// TwinCAT 3 PLC project Nepionic_OTel_IntegrationTest
// ProgramVersion: 3.1.4026.25
// libraries:
//   [Nepionic_Log], * (Nepionic)
//   Tc2_Standard, * (Beckhoff Automation GmbH)
//   Tc2_System, * (Beckhoff Automation GmbH)
//   Tc2_Utilities, * (Beckhoff Automation GmbH)
// project tree:
//   Lib/ Valve.TcPOU, FilterConfig.TcDUT, FilterSimulation.TcPOU, FilterState.TcDUT (not stored), Valve.TcPOU
//   Programs/ Main.TcPOU
//   Tasks/ PlcTask.TcTTO
// real-time tasks:
//   TASK PlcTask: cycle T#10ms, priority 20, ADS port 350

CONFIGURATION Nepionic_OTel_IntegrationTest
    RESOURCE PLC ON TwinCAT3
        TASK PlcTask(INTERVAL := T#10ms, PRIORITY := 20);
        PROGRAM Main WITH PlcTask : Main;
    END_RESOURCE
END_CONFIGURATION

// ---- Lib/FilterConfig.TcDUT
/// Configuration parameters for the sand filter simulation.
/// All *_s fields are in simulated seconds.
/// Real elapsed time = simulated_time / time_scale.
TYPE FilterConfig :
STRUCT
    /// Nominal (clean-filter) differential pressure across the filter bank (bar).
    dp_nominal_bar         : LREAL := 0.15;
    /// Differential pressure that triggers a backwash cycle (bar).
    dp_trigger_bar         : LREAL := 0.80;
    /// Theoretical maximum differential pressure of a fully blocked filter (bar).
    dp_max_bar             : LREAL := 1.40;
    /// Nominal pump flow rate during normal two-module filtering (L/min).
    flow_nominal_lpm       : LREAL := 500.0;
    /// Reduced pump flow rate during backwash — one module out of service (L/min).
    flow_backwash_lpm      : LREAL := 340.0;
    /// Static inlet pressure at nominal flow with a clean filter (bar).
    pressure_inlet_bar     : LREAL := 2.50;
    /// Simulated time for the filter to block from clean to dp_trigger_bar (seconds).
    blockage_time_s        : LREAL := 300.0;
    /// Duration of each individual module backwash phase (simulated seconds).
    backwash_duration_s    : LREAL := 30.0;
    /// Settling delay between Module A backwash end and Module B backwash start
    /// (simulated seconds).
    inter_backwash_delay_s : LREAL := 5.0;
    /// Post-backwash settling period before resuming normal filtering
    /// (simulated seconds).
    post_backwash_settle_s : LREAL := 10.0;
    /// Simulation time scale: simulated seconds that pass per real second.
    /// 10.0 means the filter blocks in blockage_time_s/10 real seconds.
    time_scale             : LREAL := 10.0;
    /// PLC task cycle time (ms) — used for per-scan blockage accumulation.
    cycle_time_ms          : LREAL := 10.0;
END_STRUCT
END_TYPE

// ---- Programs/Main.TcPOU
/// Integration test: self-cleaning reverse-flow sand filter.
///
/// Wires the FilterSimulation to the Nepionic Log + Metrics OTel bridge.
/// Both the log ring and metric ring are exposed as ADS symbols — point
/// the otelcol-ads collector at:
///   Logs    : Main.log_appender.ring
///   Metrics : Main.metric_ring
PROGRAM Main
VAR
    // ── OTel log backend ───────────────────────────────────────────────────────
    log_appender : Nepionic_Log_OTel.OTelLogAppender;

    // ── OTel metrics backend ───────────────────────────────────────────────────
    metric_core : Nepionic_Metrics_OTel.OTelMetricCore;

    // ── Application logger ─────────────────────────────────────────────────────
    logger : Nepionic_Log.DefaultLogger('SandFilter.Controller');

    // ── Filter simulation ──────────────────────────────────────────────────────
    config : FilterConfig;    // Uses DUT default values; tune at runtime.
    sim : FilterSimulation;

    // ── Metric publish interval (real time, independent of sim time_scale) ─────
    metric_timer : TON;

    // ── One-shot initialisation guard ─────────────────────────────────────────
    initialised : BOOL;

    // ── Metric attribute scratch buffers ──────────────────────────────────────
    m_attrs : ARRAY[0..4] OF Nepionic_Metrics.MetricAttribute;
    m_empty : ARRAY[0..4] OF Nepionic_Metrics.MetricAttribute;
	
	trigger_div_zero : BOOL;
	_div_zero : FLOAT;
	
	heartbeat_timer : TOn;
END_VAR

// ── One-time initialisation ───────────────────────────────────────────────────
IF NOT initialised THEN
    Nepionic_Log.GetLogManager().Register(log_appender);
    initialised := TRUE;
    logger.Info('Sand filter OTel integration test initialised');
END_IF

// ── Run filter simulation ─────────────────────────────────────────────────────
sim(Config := config);

// ── Log on state-transition events ───────────────────────────────────────────
// DP threshold crossed — backwash is about to begin.
IF sim.EvFilterBlocked THEN
    logger
        .WithAttribute('state', 'Filtering')
        .Warning('Differential pressure exceeded backwash threshold - scheduling backwash cycle');
END_IF

// Module A backwash valve just opened.
IF sim.EvBackwashStartedA THEN
    logger
        .WithAttribute('module', 'A')
        .WithAttribute('valve',  'reverse_flow_A')
        .Info('Backwash started - Module A reverse-flow valve open, waste port active');
END_IF

// Module B backwash valve just opened.
IF sim.EvBackwashStartedB THEN
    logger
        .WithAttribute('module', 'B')
        .WithAttribute('valve',  'reverse_flow_B')
        .Info('Backwash started - Module B reverse-flow valve open, waste port active');
END_IF

// Both modules cleaned; filter bank back in service.
IF sim.EvBackwashComplete THEN
    logger
        .WithAttribute('cycles_completed', UDINT_TO_STRING(sim.BackwashCycles))
        .Info('Full backwash cycle complete - both modules clean, differential pressure at nominal');
END_IF

// ── Publish metrics every second (real time) ──────────────────────────────────
metric_timer(IN := TRUE, PT := T#1S);
IF metric_timer.Q THEN
    metric_timer(IN := FALSE); // reset for next interval

    // Pump flow
    metric_core.Record(
        'filter.flow_rate', 'L/min',
        sim.PumpFlowLpm,
        Nepionic_Metrics.MetricKind.Gauge, m_empty, 0);

    // Filter bank pressures
    metric_core.Record(
        'filter.pressure.inlet', 'bar',
        sim.PressureInletBar,
        Nepionic_Metrics.MetricKind.Gauge, m_empty, 0);

    metric_core.Record(
        'filter.pressure.outlet', 'bar',
        sim.PressureOutletBar,
        Nepionic_Metrics.MetricKind.Gauge, m_empty, 0);

    metric_core.Record(
        'filter.pressure.differential', 'bar',
        sim.DpBar,
        Nepionic_Metrics.MetricKind.Gauge, m_empty, 0);

    // Blockage fraction — key indicator driving the backwash trigger
    metric_core.Record(
        'filter.blockage_fraction', '1',
        sim.BlockageFraction,
        Nepionic_Metrics.MetricKind.Gauge, m_empty, 0);

    // Monotonically increasing backwash cycle counter
    metric_core.Record(
        'filter.backwash.cycles_total', '{cycles}',
        UDINT_TO_LREAL(sim.BackwashCycles),
        Nepionic_Metrics.MetricKind.Counter, m_empty, 0);

    // Per-module backwash valve state (0=closed, 1=open), labelled by module
    m_attrs[0].key := 'module'; m_attrs[0].value := 'A';
    metric_core.Record(
        'filter.valve.backwash_active', '1',
        SEL(sim.ValveAOpen, 0.0, 1.0),
        Nepionic_Metrics.MetricKind.Gauge, m_attrs, 1);

    m_attrs[0].value := 'B';
    metric_core.Record(
        'filter.valve.backwash_active', '1',
        SEL(sim.ValveBOpen, 0.0, 1.0),
        Nepionic_Metrics.MetricKind.Gauge, m_attrs, 1);
END_IF

IF trigger_div_zero THEN
	trigger_div_zero := FALSE;
	_div_zero := 1 / _div_zero;
END_IF

heartbeat_timer(In := NOT heartbeat_timer.Q, PT := T#5S);
IF heartbeat_timer.Q THEN
    log_appender.Heartbeat();
	metric_core.Heartbeat();
END_IF

END_PROGRAM

// ---- Lib/FilterSimulation.TcPOU
/// Simulated reverse-flow self-cleaning sand filter with two filter modules.
///
/// Physical model
/// ─────────────
/// Filtering (normal):
///   Pump → Inlet → [Module A + Module B in parallel] → Outlet
///   Differential pressure rises as both modules accumulate blockage.
///
/// Backwash (Module A):
///   Clean outlet water is diverted backwards through Module A → Waste.
///   Module B carries all forward flow; DP reflects one module.
///
/// Backwash (Module B):  symmetric to Module A.
///
/// After BackwashB completes the blockage fraction is reset to zero and the
/// differential pressure returns to nominal.
///
/// Call every PLC scan and read the VAR_OUTPUT fields.
FUNCTION_BLOCK FilterSimulation
VAR_INPUT
    /// Simulation configuration (may be updated at runtime).
    Config : FilterConfig;
END_VAR
VAR_OUTPUT
    // ── Sensors ───────────────────────────────────────────────────────────────
    /// Pump flow rate (L/min).
    PumpFlowLpm         : LREAL;
    /// Filter bank inlet pressure (bar).
    PressureInletBar    : LREAL;
    /// Filter bank outlet pressure (bar).
    PressureOutletBar   : LREAL;
    /// Differential pressure across the filter bank: inlet − outlet (bar).
    DpBar               : LREAL;

    // ── Valve states ──────────────────────────────────────────────────────────
    /// TRUE when Module A reverse-flow backwash valve is open.
    ValveAOpen          : BOOL;
    /// TRUE when Module B reverse-flow backwash valve is open.
    ValveBOpen          : BOOL;

    // ── Status ────────────────────────────────────────────────────────────────
    /// Current controller state.
    State               : FilterState := FilterState.Filtering;
    /// Number of complete two-module backwash cycles executed since PLC start.
    BackwashCycles      : UDINT;
    /// Blockage fraction: 0.0 = completely clean, 1.0 = theoretical dp_max_bar.
    BlockageFraction    : LREAL;

    // ── Event pulses (TRUE for exactly one scan on the triggering transition) ─
    /// DP has just exceeded dp_trigger_bar — backwash is about to start.
    EvFilterBlocked     : BOOL;
    /// Module A backwash valve has just been opened.
    EvBackwashStartedA  : BOOL;
    /// Module B backwash valve has just been opened.
    EvBackwashStartedB  : BOOL;
    /// Full two-module backwash cycle just completed; blockage reset to zero.
    EvBackwashComplete  : BOOL;
END_VAR
VAR
    _blockage         : LREAL := 0.0;  // 0.0 (clean) → 1.0 (at dp_max_bar)
    _entry            : BOOL  := TRUE; // TRUE on the first scan of a new state
    _timer            : TON;
    _timer_pt         : TIME;
    _valveA           : Valve;
    _valveB           : Valve;
    _noise_t          : LREAL := 0.0;  // noise oscillator phase accumulator
    _noise            : LREAL;         // composite dimensionless noise signal
    _sim_dt           : LREAL;         // simulated seconds elapsed this scan
    _blockage_trigger : LREAL;         // blockage fraction that fires backwash
END_VAR

// ── Per-scan simulated timestep ──────────────────────────────────────────────
_sim_dt := Config.cycle_time_ms * 0.001 * Config.time_scale;

// Normalised blockage fraction at which dp_trigger_bar is reached.
_blockage_trigger := (Config.dp_trigger_bar - Config.dp_nominal_bar)
                   / (Config.dp_max_bar     - Config.dp_nominal_bar);

// ── Multi-frequency noise oscillator ─────────────────────────────────────────
// Phase advances at ~0.5 rad/real-second, giving a ~12-second noise period.
_noise_t := _noise_t + Config.cycle_time_ms * 0.001 * 0.5;
IF _noise_t > 628.0 THEN _noise_t := _noise_t - 628.0; END_IF
_noise := 0.015 * SIN(_noise_t)
        + 0.008 * SIN(_noise_t * 2.37 + 1.1)
        + 0.004 * SIN(_noise_t * 5.13 + 2.3);

// ── Clear event pulses ────────────────────────────────────────────────────────
EvFilterBlocked    := FALSE;
EvBackwashStartedA := FALSE;
EvBackwashStartedB := FALSE;
EvBackwashComplete := FALSE;

// ── State machine ─────────────────────────────────────────────────────────────
CASE State OF

    FilterState.Filtering:
        _valveA(Open := FALSE, Close := TRUE);
        _valveB(Open := FALSE, Close := TRUE);

        // Blockage accumulates while both modules are filtering.
        _blockage := MIN(_blockage + _sim_dt / Config.blockage_time_s, 1.0);

        // Trigger backwash when DP crosses dp_trigger_bar.
        IF _blockage >= _blockage_trigger THEN
            EvFilterBlocked := TRUE;
            State           := FilterState.BackwashA;
            _entry          := TRUE;
        END_IF

    FilterState.BackwashA:
        // Module A valve open: clean water from Module B flushes Module A to waste.
        _valveA(Open := TRUE,  Close := FALSE);
        _valveB(Open := FALSE, Close := TRUE);

        IF _entry THEN
            _entry             := FALSE;
            EvBackwashStartedA := TRUE;
            _timer(IN := FALSE, PT := T#0S); // reset
        ELSE
            _timer_pt := UDINT_TO_TIME(LREAL_TO_UDINT(
                Config.backwash_duration_s / Config.time_scale * 1000.0));
            _timer(IN := TRUE, PT := _timer_pt);
            IF _timer.Q THEN
                _timer(IN := FALSE, PT := T#0S);
                State  := FilterState.PauseBetween;
                _entry := TRUE;
            END_IF
        END_IF

    FilterState.PauseBetween:
        // Both valves closed; brief settling before opening Module B valve.
        _valveA(Open := FALSE, Close := TRUE);
        _valveB(Open := FALSE, Close := TRUE);

        IF _entry THEN
            _entry := FALSE;
            _timer(IN := FALSE, PT := T#0S);
        ELSE
            _timer_pt := UDINT_TO_TIME(LREAL_TO_UDINT(
                Config.inter_backwash_delay_s / Config.time_scale * 1000.0));
            _timer(IN := TRUE, PT := _timer_pt);
            IF _timer.Q THEN
                _timer(IN := FALSE, PT := T#0S);
                State  := FilterState.BackwashB;
                _entry := TRUE;
            END_IF
        END_IF

    FilterState.BackwashB:
        // Module B valve open: clean water from Module A flushes Module B to waste.
        _valveA(Open := FALSE, Close := TRUE);
        _valveB(Open := TRUE,  Close := FALSE);

        IF _entry THEN
            _entry             := FALSE;
            EvBackwashStartedB := TRUE;
            _timer(IN := FALSE, PT := T#0S);
        ELSE
            _timer_pt := UDINT_TO_TIME(LREAL_TO_UDINT(
                Config.backwash_duration_s / Config.time_scale * 1000.0));
            _timer(IN := TRUE, PT := _timer_pt);
            IF _timer.Q THEN
                _timer(IN := FALSE, PT := T#0S);
                _blockage := 0.0;  // Both modules cleaned — reset blockage.
                State     := FilterState.PostBackwash;
                _entry    := TRUE;
            END_IF
        END_IF

    FilterState.PostBackwash:
        // Both valves closed; pressure and flow settle before resuming filtering.
        _valveA(Open := FALSE, Close := TRUE);
        _valveB(Open := FALSE, Close := TRUE);

        IF _entry THEN
            _entry             := FALSE;
            EvBackwashComplete := TRUE;
            BackwashCycles     := BackwashCycles + 1;
            _timer(IN := FALSE, PT := T#0S);
        ELSE
            _timer_pt := UDINT_TO_TIME(LREAL_TO_UDINT(
                Config.post_backwash_settle_s / Config.time_scale * 1000.0));
            _timer(IN := TRUE, PT := _timer_pt);
            IF _timer.Q THEN
                _timer(IN := FALSE, PT := T#0S);
                State  := FilterState.Filtering;
                _entry := TRUE;
            END_IF
        END_IF

END_CASE

// ── Valve outputs ─────────────────────────────────────────────────────────────
ValveAOpen       := _valveA.IsOpen;
ValveBOpen       := _valveB.IsOpen;
BlockageFraction := _blockage;

// ── Differential pressure ─────────────────────────────────────────────────────
// During backwash one module is bypassed; DP reflects the remaining clean module
// (slightly above nominal due to full flow through half the filter area).
// During filtering the DP rises linearly with blockage, noised for realism.
IF    State = FilterState.BackwashA
   OR State = FilterState.PauseBetween
   OR State = FilterState.BackwashB THEN
    DpBar := Config.dp_nominal_bar * 1.25 * (1.0 + _noise);
ELSE
    DpBar := Config.dp_nominal_bar
           + _blockage * (Config.dp_max_bar - Config.dp_nominal_bar);
    DpBar := DpBar * (1.0 + _noise);
END_IF
DpBar := MAX(DpBar, 0.0);

// ── Inlet pressure ────────────────────────────────────────────────────────────
// The pump works slightly harder as filter resistance increases.
PressureInletBar := Config.pressure_inlet_bar
                  * (1.0 + 0.04 * _blockage)
                  * (1.0 + _noise * 0.5);

// ── Outlet pressure ───────────────────────────────────────────────────────────
PressureOutletBar := PressureInletBar - DpBar;

// ── Pump flow ─────────────────────────────────────────────────────────────────
// Flow drops during backwash: only one module in forward service, plus the
// backwash return path consumes part of the output.
IF State = FilterState.BackwashA OR State = FilterState.BackwashB THEN
    PumpFlowLpm := Config.flow_backwash_lpm * (1.0 + _noise * 0.3);
ELSE
    PumpFlowLpm := Config.flow_nominal_lpm  * (1.0 + _noise * 0.3);
END_IF
PumpFlowLpm := MAX(PumpFlowLpm, 0.0);

END_FUNCTION_BLOCK

// ---- Lib/Valve.TcPOU
/// Simulated latching actuated valve.
/// Open/Close are momentary command inputs; position is retained between scans.
/// Open takes priority over Close.
FUNCTION_BLOCK Valve
VAR_INPUT
    Open  : BOOL; /// Momentary command: open the valve.
    Close : BOOL; /// Momentary command: close the valve.
END_VAR
VAR_OUTPUT
    IsOpen   : BOOL; /// TRUE when valve is in the fully open position.
    IsClosed : BOOL; /// TRUE when valve is in the fully closed position.
END_VAR
VAR
    _open : BOOL := FALSE;
END_VAR

// Open wins over Close.
IF Open THEN
    _open := TRUE;
ELSIF Close THEN
    _open := FALSE;
END_IF

IsOpen   := _open;
IsClosed := NOT _open;

END_FUNCTION_BLOCK

// ---- Lib/Valve.TcPOU
/// Simulated latching actuated valve.
/// Open/Close are momentary command inputs; position is retained between scans.
/// Open takes priority over Close.
FUNCTION_BLOCK Valve
VAR_INPUT
    Open  : BOOL; /// Momentary command: open the valve.
    Close : BOOL; /// Momentary command: close the valve.
END_VAR
VAR_OUTPUT
    IsOpen   : BOOL; /// TRUE when valve is in the fully open position.
    IsClosed : BOOL; /// TRUE when valve is in the fully closed position.
END_VAR
VAR
    _open : BOOL := FALSE;
END_VAR

// Open wins over Close.
IF Open THEN
    _open := TRUE;
ELSIF Close THEN
    _open := FALSE;
END_IF

IsOpen   := _open;
IsClosed := NOT _open;

END_FUNCTION_BLOCK
